FUNCTION_BLOCK FB_SecondOrder
VAR_INPUT
END_VAR
VAR_OUTPUT
END_VAR
VAR CONSTANT
	order : INT := 2;
END_VAR

METHOD Determinant2x2 : BOOL
VAR_INPUT
	ptrDeterminant	: POINTER TO LREAL;
	ptrMatrix		: POINTER TO ARRAY[1..2,1..2] OF LREAL;	
END_VAR
ptrDeterminant^ := ptrMatrix^[2,2]*ptrMatrix^[1,1] - ptrMatrix^[1,2]*ptrMatrix^[2,1];
END_METHOD

METHOD Determinant3x3 : BOOL
VAR_INPUT
	ptrDeterminant	: POINTER TO LREAL;
	ptrMatrix		: POINTER TO ARRAY[1..3,1..3] OF LREAL;
END_VAR
VAR
	Matrix3x3		: ARRAY[1..3,1..3] OF LREAL;
	Element1		: LREAL;
	Element2		: LREAL;
	RowMultiplier	: LREAL;
	i				: INT;
	j				: INT;
	row 			: INT;
	currentRow		: INT;
	temp			: LREAL;
	Swap			: BOOL;
	index			: INT;
	found			: BOOL;
END_VAR
Matrix3x3 := ptrMatrix^;
Swap := FALSE;
FOR index := 1 TO order DO
	IF Matrix3x3[index,index] = 0 THEN
		found := FALSE;
		FOR i:=index+1 TO 3 DO
			IF Matrix3x3[index,i] <> 0 THEN
				row := i;
				found := TRUE;
				EXIT;
			END_IF
		END_FOR
		// swap current row with found row
		IF found THEN
			FOR i := 1 TO order+1 DO
				temp := Matrix3x3[i,index];
				Matrix3x3[i,index] := Matrix3x3[i,row];
				Matrix3x3[i,row] := temp;
			END_FOR
			Swap := NOT Swap;
		ELSE
			ptrDeterminant^ := 0;
			Determinant3x3 := FALSE;
			RETURN;
		END_IF
	END_IF
	
	FOR j := index+1 TO order+1 DO
		Element1 := Matrix3x3[index,index];
		Element2 := Matrix3x3[index,j];
		IF Element2 <> 0 THEN
			RowMultiplier := Element2/Element1;
			FOR i := 1 TO order+1 DO
				Matrix3x3[i,j] := Matrix3x3[i,j] - RowMultiplier*Matrix3x3[i,index];
			END_FOR
		END_IF
	END_FOR
END_FOR

ptrDeterminant^ := 1;
FOR i := 1 TO order+1 DO
	ptrDeterminant^ := ptrDeterminant^ * Matrix3x3[i,i];
END_FOR

IF Swap THEN
	ptrDeterminant^ := ptrDeterminant^ * (-1);
END_IF	
Determinant3x3 := TRUE;
END_METHOD

METHOD Determinant4x4 : BOOL
VAR_INPUT
	ptrDeterminant	: POINTER TO LREAL;
	ptrMatrix		: POINTER TO ARRAY[1..4,1..4] OF LREAL;
END_VAR
VAR
	Matrix4x4		: ARRAY[1..4,1..4] OF LREAL;
	Element1		: LREAL;
	Element2		: LREAL;
	RowMultiplier	: LREAL;
	i				: INT;
	j				: INT;
	row 			: INT;
	currentRow		: INT;
	temp			: LREAL;
	Swap			: BOOL;
	index			: INT;
	found			: BOOL;
END_VAR
Matrix4x4 := ptrMatrix^;
Swap := FALSE;
FOR index := 1 TO 3 DO
	IF Matrix4x4[index,index] = 0 THEN
		found := FALSE;
		FOR i:=index+1 TO 4 DO
			IF Matrix4x4[index,i] <> 0 THEN
				row := i;
				found := TRUE;
				EXIT;
			END_IF
		END_FOR
		// swap current row with found row
		IF found THEN
			FOR i := 1 TO 4 DO
				temp := Matrix4x4[i,index];
				Matrix4x4[i,index] := Matrix4x4[i,row];
				Matrix4x4[i,row] := temp;
			END_FOR
			Swap := NOT Swap;
		ELSE
			ptrDeterminant^ := 0;
			Determinant4x4 := FALSE;
			RETURN;
		END_IF
	END_IF
	
	FOR j := index+1 TO 4 DO
		Element1 := Matrix4x4[index,index];
		Element2 := Matrix4x4[index,j];
		IF Element2 <> 0 THEN
			RowMultiplier := Element2/Element1;
			FOR i := 1 TO 4 DO
				Matrix4x4[i,j] := Matrix4x4[i,j] - RowMultiplier*Matrix4x4[i,index];
			END_FOR
		END_IF
	END_FOR
END_FOR

ptrDeterminant^ := 1;
FOR i := 1 TO 4 DO
	ptrDeterminant^ := ptrDeterminant^ * Matrix4x4[i,i];
END_FOR

IF Swap THEN
	ptrDeterminant^ := ptrDeterminant^ * (-1);
END_IF	
Determinant4x4 := TRUE;
END_METHOD

METHOD Determinant5x5 : BOOL
VAR_INPUT
	ptrDeterminant	: POINTER TO LREAL;
	ptrMatrix		: POINTER TO ARRAY[1..5,1..5] OF LREAL;
END_VAR
VAR
	Matrix5x5		: ARRAY[1..5,1..5] OF LREAL;
	Element1		: LREAL;
	Element2		: LREAL;
	RowMultiplier	: LREAL;
	i				: INT;
	j				: INT;
	row 			: INT;
	currentRow		: INT;
	temp			: LREAL;
	Swap			: BOOL;
	index			: INT;
	found			: BOOL;
END_VAR
Matrix5x5 := ptrMatrix^;
Swap := FALSE;
FOR index := 1 TO 4 DO
	IF Matrix5x5[index,index] = 0 THEN
		found := FALSE;
		FOR i:=index+1 TO 5 DO
			IF Matrix5x5[index,i] <> 0 THEN
				row := i;
				found := TRUE;
				EXIT;
			END_IF
		END_FOR
		// swap current row with found row
		IF found THEN
			FOR i := 1 TO 5 DO
				temp := Matrix5x5[i,index];
				Matrix5x5[i,index] := Matrix5x5[i,row];
				Matrix5x5[i,row] := temp;
			END_FOR
			Swap := NOT Swap;
		ELSE
			ptrDeterminant^ := 0;
			Determinant5x5 := FALSE;
			RETURN;
		END_IF
	END_IF
	
	FOR j := index+1 TO 5 DO
		Element1 := Matrix5x5[index,index];
		Element2 := Matrix5x5[index,j];
		IF Element2 <> 0 THEN
			RowMultiplier := Element2/Element1;
			FOR i := 1 TO 5 DO
				Matrix5x5[i,j] := Matrix5x5[i,j] - RowMultiplier*Matrix5x5[i,index];
			END_FOR
		END_IF
	END_FOR
END_FOR

ptrDeterminant^ := 1;
FOR i := 1 TO 5 DO
	ptrDeterminant^ := ptrDeterminant^ * Matrix5x5[i,i];
END_FOR

IF Swap THEN
	ptrDeterminant^ := ptrDeterminant^ * (-1);
END_IF	
Determinant5x5 := TRUE;
END_METHOD

METHOD FindCoefficients : BOOL
VAR_INPUT
	xValues		: POINTER TO ARRAY[1..GVL.NumberVisionPoints] OF LREAL;
	yValues		: POINTER TO ARRAY[1..GVL.NumberVisionPoints] OF LREAL;
	Coefficients: POINTER TO ARRAY[1..3] OF LREAL;
END_VAR
VAR_INST 
	xMatrix		: ARRAY[1..3, 1..GVL.NumberVisionPoints] OF LREAL;
	xTMatrix	: ARRAY[1..GVL.NumberVisionPoints, 1..3] OF LREAL; 
	xTxMatrix	: ARRAY[1..3,1..3] OF LREAL;
	xTxInverse	: ARRAY[1..3,1..3] OF LREAL;
	xTyMatrix	: ARRAY[1..3] OF LREAL;
	i			: INT;
	j			: INT;
	k			: INT;
	DotProduct	: LREAL;
END_VAR
// fill out x matrix
// fill out transpose of x matrix
FOR i := 1 TO order+1 DO	// column
	FOR j := 1 TO GVL.NumberVisionPoints DO
		xMatrix[i,j] := EXPT((xValues^[j]),(i-1));	
		xTMatrix[j,i] := xMatrix[i,j];
	END_FOR
END_FOR

// fill out xT * x 
FOR i := 1 TO order+1 DO		// rows
	FOR j := 1 TO order+1 DO	
		DotProduct := 0;
		FOR k := 1 TO GVL.NumberVisionPoints DO
			DotProduct := DotProduct + xTMatrix[k,i]*xMatrix[j,k];
		END_FOR
		xTxMatrix[j,i] := DotProduct;
	END_FOR
END_FOR

// find out the inverse of xT*x
Inverse(ptrMatrix := ADR(xTxMatrix), ptrInverse := ADR(xTxInverse));

// multiple xT*y
FOR i := 1 TO order+1 DO 
	DotProduct := 0;
	FOR j := 1 TO GVL.NumberVisionPoints DO
		DotProduct := DotProduct + xTMatrix[j,i] * yValues^[j];
	END_FOR
	xTyMatrix[i] := DotProduct;
END_FOR

// multiply xTxInverse by xTy
FOR i := 1 TO order+1 DO
	DotProduct := 0;
	FOR j := 1 TO order+1 DO
		DotProduct := DotProduct + xTxInverse[j,i]*xTyMatrix[j];
	END_FOR
	Coefficients^[i] := DotProduct;
END_FOR
END_METHOD

METHOD FindPeak : LREAL
VAR_INPUT
	xValues		: POINTER TO ARRAY[1..GVL.NumberVisionPoints] OF LREAL;
	yValues		: POINTER TO ARRAY[1..GVL.NumberVisionPoints] OF LREAL;
	xPeak		: POINTER TO LREAL;
END_VAR
VAR
	Coefficients: ARRAY[1..3] OF LREAL;	
	a			: LREAL;
	b			: LREAL;
END_VAR
FindCoefficients(xValues := xValues, yValues := yValues, Coefficients := ADR(Coefficients));
a := Coefficients[3];
b := Coefficients[2];
xPeak^ := -b/(2*a);
END_METHOD

METHOD Inverse : BOOL
VAR_INPUT
	ptrMatrix		: POINTER TO ARRAY[1..3,1..3] OF LREAL;
	ptrInverse		: POINTER TO ARRAY[1..3,1..3] OF LREAL;
END_VAR
VAR_INST
	Matrix3x3		: ARRAY[1..3,1..3] OF LREAL;
	Determinant		: LREAL;
	Matrix			: ARRAY[1..3,1..3] OF LREAL; // matrix of minors
	Matrix2x2		: ARRAY[1..2,1..2] OF LREAL;
	_Cofactor		: LREAL;
	i				: INT;
	j				: INT;
	SignRow			: BOOL;
	SignColumn		: BOOL;
END_VAR
Matrix3x3 := ptrMatrix^;

IF Determinant3x3(ptrDeterminant := ADR(Determinant), ptrMatrix := ptrMatrix) THEN
	Determinant := 1 / Determinant;

	// matrix of minors
	// column 1:
	Matrix2x2[1,1] := Matrix3x3[2,2];
	Matrix2x2[1,2] := Matrix3x3[2,3];
	Matrix2x2[2,1] := Matrix3x3[3,2];
	Matrix2x2[2,2] := Matrix3x3[3,3];
	Determinant2x2(ADR(Matrix[1,1]), ADR(Matrix2x2));

	Matrix2x2[1,1] := Matrix3x3[2,1];
	Matrix2x2[1,2] := Matrix3x3[2,3];
	Matrix2x2[2,1] := Matrix3x3[3,1];
	Matrix2x2[2,2] := Matrix3x3[3,3];
	Determinant2x2(ADR(Matrix[1,2]), ADR(Matrix2x2));

	Matrix2x2[1,1] := Matrix3x3[2,1];
	Matrix2x2[1,2] := Matrix3x3[2,2];
	Matrix2x2[2,1] := Matrix3x3[3,1];
	Matrix2x2[2,2] := Matrix3x3[3,2];
	Determinant2x2(ADR(Matrix[1,3]), ADR(Matrix2x2));
	
	// column 2:
	Matrix2x2[1,1] := Matrix3x3[1,2];
	Matrix2x2[1,2] := Matrix3x3[1,3];
	Matrix2x2[2,1] := Matrix3x3[3,2];
	Matrix2x2[2,2] := Matrix3x3[3,3];
	Determinant2x2(ADR(Matrix[2,1]), ADR(Matrix2x2));

	Matrix2x2[1,1] := Matrix3x3[1,1];
	Matrix2x2[1,2] := Matrix3x3[1,3];
	Matrix2x2[2,1] := Matrix3x3[3,1];
	Matrix2x2[2,2] := Matrix3x3[3,3];
	Determinant2x2(ADR(Matrix[2,2]), ADR(Matrix2x2));

	Matrix2x2[1,1] := Matrix3x3[1,1];
	Matrix2x2[1,2] := Matrix3x3[1,2];
	Matrix2x2[2,1] := Matrix3x3[3,1];
	Matrix2x2[2,2] := Matrix3x3[3,2];
	Determinant2x2(ADR(Matrix[2,3]), ADR(Matrix2x2));

	// column 3:
	Matrix2x2[1,1] := Matrix3x3[1,2];
	Matrix2x2[1,2] := Matrix3x3[1,3];
	Matrix2x2[2,1] := Matrix3x3[2,2];
	Matrix2x2[2,2] := Matrix3x3[2,3];
	Determinant2x2(ADR(Matrix[3,1]), ADR(Matrix2x2));

	Matrix2x2[1,1] := Matrix3x3[1,1];
	Matrix2x2[1,2] := Matrix3x3[1,3];
	Matrix2x2[2,1] := Matrix3x3[2,1];
	Matrix2x2[2,2] := Matrix3x3[2,3];
	Determinant2x2(ADR(Matrix[3,2]), ADR(Matrix2x2));

	Matrix2x2[1,1] := Matrix3x3[1,1];
	Matrix2x2[1,2] := Matrix3x3[1,2];
	Matrix2x2[2,1] := Matrix3x3[2,1];
	Matrix2x2[2,2] := Matrix3x3[2,2];
	Determinant2x2(ADR(Matrix[3,3]), ADR(Matrix2x2));
	
	// switch the signs	
	SignRow := TRUE;
	SignColumn := TRUE;
	FOR i := 1 TO order+1 DO
		FOR j := 1 TO order+1 DO
			IF NOT SignRow THEN
				Matrix[i,j] := (-1) * Matrix[i,j];
			END_IF
			SignRow := NOT SignRow;
		END_FOR
		SignColumn := NOT SignColumn;
		SignRow := SignColumn;
	END_FOR
	// transpose 
	Transpose(ADR(Matrix),ptrInverse);
	FOR i := 1 TO order+1 DO
		FOR j := 1 TO order+1 DO
			ptrInverse^[i,j] := Determinant * ptrInverse^[i,j];
		END_FOR
	END_FOR
	
	Inverse := TRUE;
ELSE
	Inverse := FALSE;
END_IF
END_METHOD

METHOD Transpose : BOOL
VAR_INPUT
	ptrMatrix		: POINTER TO ARRAY[1..3,1..3] OF LREAL;
	ptrTranspose	: POINTER TO ARRAY[1..3,1..3] OF LREAL;
END_VAR
VAR
	i				: INT;
	j				: INT;
END_VAR
FOR i := 1 TO order+1 DO
	FOR j := 1 TO order+1 DO
		ptrTranspose^[j,i] := ptrMatrix^[i,j];
	END_FOR
END_FOR
END_METHOD

END_FUNCTION_BLOCK

(* stored: Version 1.1.0.1, ProductVersion 3.1.4024.3
   POU FB_SecondOrder: Id {b4b11a2b-7815-44ba-962d-86f46f681442}, SpecialFunc None
   Method Determinant2x2: Id {de06f8cf-8e05-4aa0-b287-74a9c4a12efe}
   Method Determinant3x3: Id {5d4f1ac7-18eb-4a3b-b400-a829312f425e}
   Method Determinant4x4: Id {387dacad-3851-4770-a623-c0fe25f723af}
   Method Determinant5x5: Id {be49c93a-13e0-4050-8bcb-2474a1928cff}
   Method FindCoefficients: Id {4373551e-02c3-4dda-8eea-6b9f556fb716}
   Method FindPeak: Id {d9ecad1c-5ca2-4f7b-b4b8-c760752453c6}
   Method Inverse: Id {8387734f-b73e-475d-9575-67f8de8e2998}
   Method Transpose: Id {1e5f094d-9496-4290-b4a9-70d0c7b657b5} *)
